(* Schneider Machine Expert - Basic project From-A-to-B-SetAndReset, file version 2.7.0.0 *)
(* ProjectInformations: Name=Nuevo proyecto *)

HARDWARE
  Cpu 0: TM221M16R/G
  EthernetConfiguration: NetworkName=M221, IpAllocationMode=FixedAddress, IpAddress=0.0.0.0, SubnetMask=0.0.0.0
  SerialLineConfiguration: Baud=Baud19200, Parity=ParityEven, DataBits=DataBits8, StopBits=StopBits1, PhysicalMedium=PhysicalMediumRs485, TransmissionMode=TransmissionModeModbusRtu, SlaveId=1, Addressing=SlaveAddressing
  MastTask: UsePeriodScanMode=false, PeriodScan=100
  FastTask: Period=255
  CpuBehavior: StartingMode=StartAsPreviousState, AutoSaveRamOnEeprom=true, WatchdogPeriod=250

SYMBOLS  (address, symbol, comment, settings)
  %M0         "Sensor A"
  %M1         "Sensor B"
  %M3         "Conveyor"

POU Nuevo POU
  (* SectionNumber=1 *)

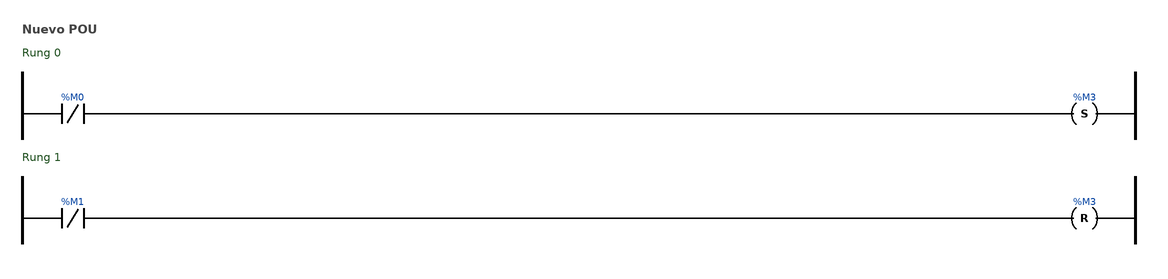

// Rung 0
  LDN %M0
  S %M3
  // as ST:
  //   IF NOT %M0 THEN %M3 := TRUE; END_IF;

// Rung 1
  LDN %M1
  R %M3
  // as ST:
  //   IF NOT %M1 THEN %M3 := FALSE; END_IF;
